(* Logix 5000 project; controller Brake_System vendor 1 type 14 code 242 rev 32.11; software revision 32.00 *)

TASK MainTask (continuous, watchdog 500 ms) : MainProgram
TASK SafetyTask (periodic, rate 20 ms, priority 10, watchdog 20 ms, safety) : SafetyProgram

MODULES
   Local : vendor 1 type 14 code 242 (5069 0, rev 32.11)
END_MODULES

PROGRAM MainProgram   (* main routine MainRoutine *)

ROUTINE MainRoutine   (* ladder *)
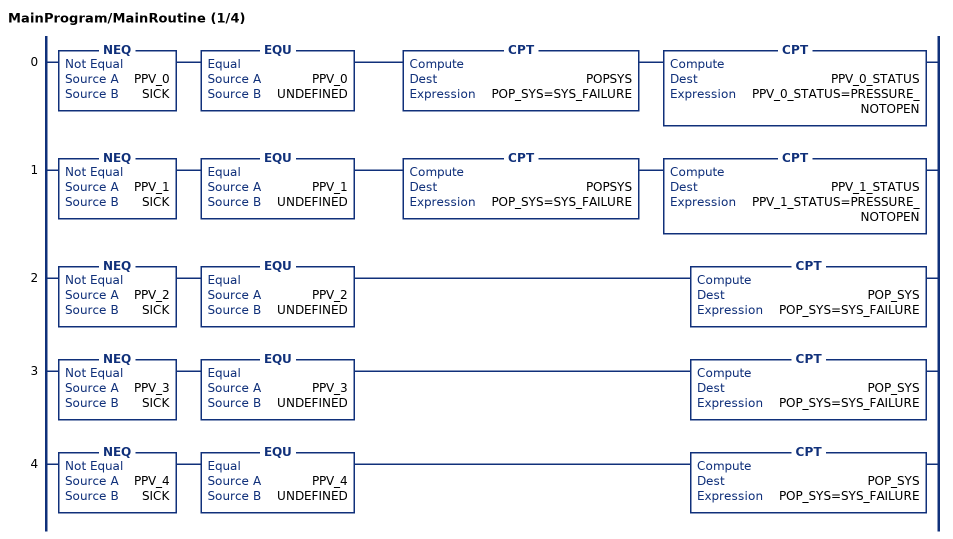
   0: NEQ(PPV_0,SICK)EQU(PPV_0,UNDEFINED)CPT(POPSYS,POP_SYS=SYS_FAILURE)CPT(PPV_0_STATUS,PPV_0_STATUS=PRESSURE_NOTOPEN);
   1: NEQ(PPV_1,SICK)EQU(PPV_1,UNDEFINED)CPT(POPSYS,POP_SYS=SYS_FAILURE)CPT(PPV_1_STATUS,PPV_1_STATUS=PRESSURE_NOTOPEN);
   2: NEQ(PPV_2,SICK)EQU(PPV_2,UNDEFINED)CPT(POP_SYS,POP_SYS=SYS_FAILURE);
   3: NEQ(PPV_3,SICK)EQU(PPV_3,UNDEFINED)CPT(POP_SYS,POP_SYS=SYS_FAILURE);
   4: NEQ(PPV_4,SICK)EQU(PPV_4,UNDEFINED)CPT(POP_SYS,POP_SYS=SYS_FAILURE);
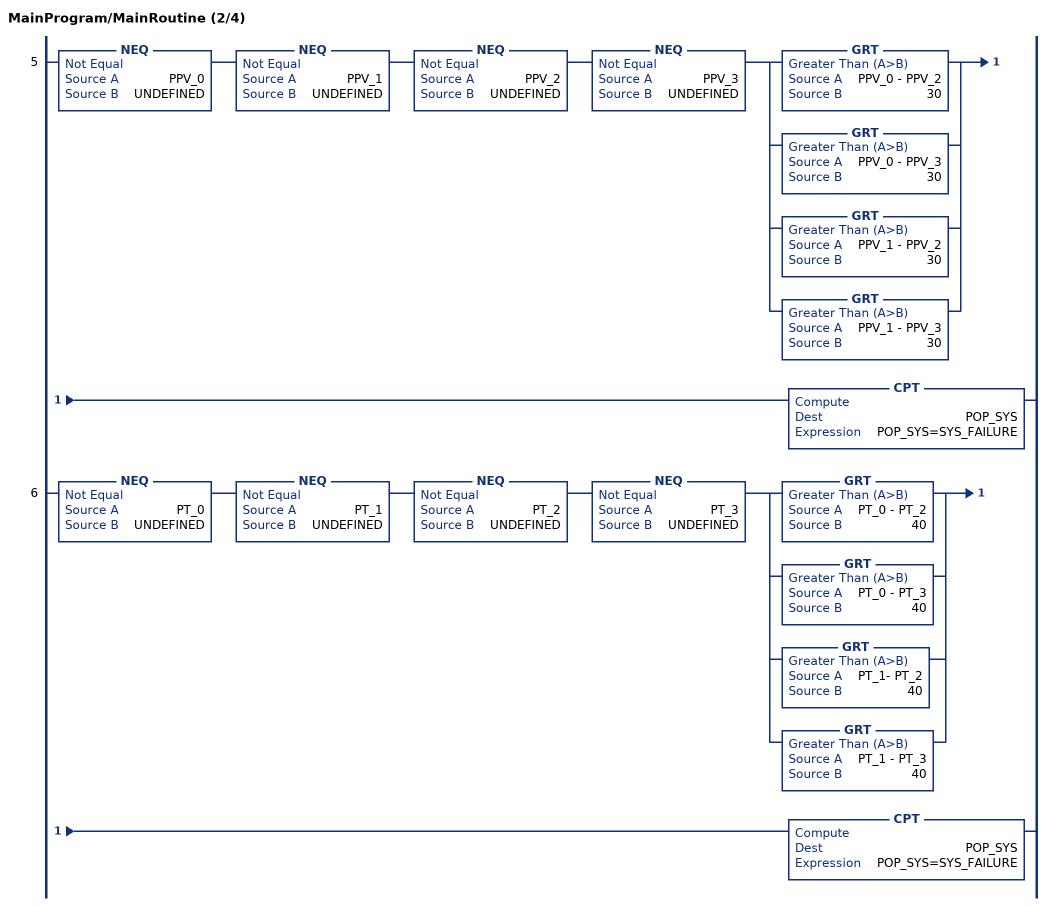
   5: NEQ(PPV_0,UNDEFINED)NEQ(PPV_1,UNDEFINED)NEQ(PPV_2,UNDEFINED)NEQ(PPV_3,UNDEFINED)[GRT(PPV_0 - PPV_2,30) ,GRT(PPV_0 - PPV_3,30) ,GRT(PPV_1 - PPV_2,30) ,GRT(PPV_1 - PPV_3,30) ]CPT(POP_SYS,POP_SYS=SYS_FAILURE);
   6: NEQ(PT_0,UNDEFINED)NEQ(PT_1,UNDEFINED)NEQ(PT_2,UNDEFINED)NEQ(PT_3,UNDEFINED)[GRT(PT_0 - PT_2,40) ,GRT(PT_0 - PT_3,40) ,GRT(PT_1- PT_2,40) ,GRT(PT_1 - PT_3,40) ]CPT(POP_SYS,POP_SYS=SYS_FAILURE);
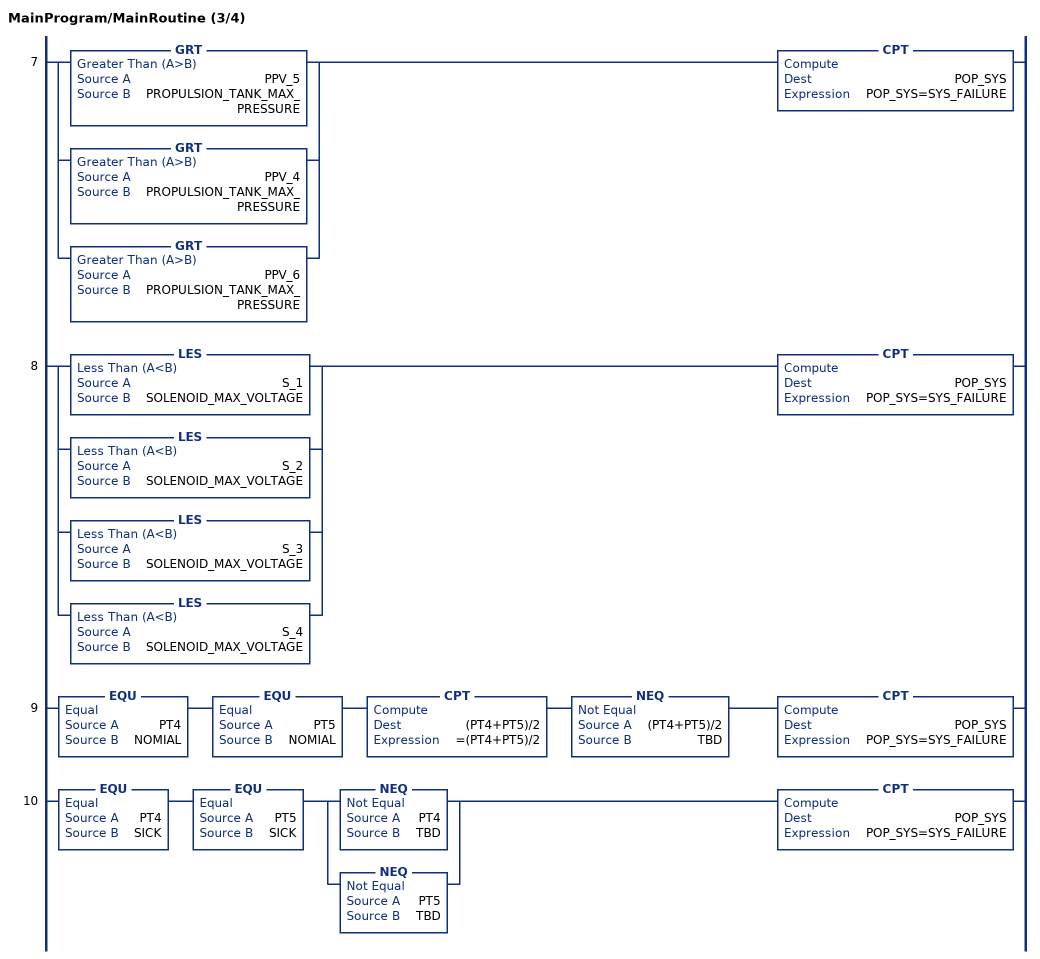
   7: [GRT(PPV_5,PROPULSION_TANK_MAX_PRESSURE) ,GRT(PPV_4,PROPULSION_TANK_MAX_PRESSURE) ,GRT(PPV_6,PROPULSION_TANK_MAX_PRESSURE) ]CPT(POP_SYS,POP_SYS=SYS_FAILURE);
   8: [LES(S_1,SOLENOID_MAX_VOLTAGE) ,LES(S_2,SOLENOID_MAX_VOLTAGE) ,LES(S_3,SOLENOID_MAX_VOLTAGE) ,LES(S_4,SOLENOID_MAX_VOLTAGE) ]CPT(POP_SYS,POP_SYS=SYS_FAILURE);
   9: EQU(PT4,NOMIAL)EQU(PT5,NOMIAL)CPT((PT4+PT5)/2,=(PT4+PT5)/2)NEQ((PT4+PT5)/2,TBD)CPT(POP_SYS,POP_SYS=SYS_FAILURE);
   10: EQU(PT4,SICK)EQU(PT5,SICK)[NEQ(PT4,TBD) ,NEQ(PT5,TBD) ]CPT(POP_SYS,POP_SYS=SYS_FAILURE);
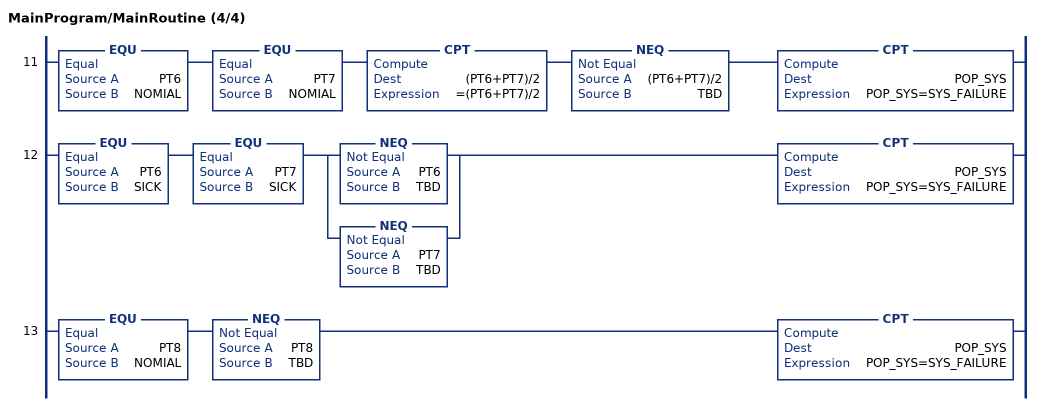
   11: EQU(PT6,NOMIAL)EQU(PT7,NOMIAL)CPT((PT6+PT7)/2,=(PT6+PT7)/2)NEQ((PT6+PT7)/2,TBD)CPT(POP_SYS,POP_SYS=SYS_FAILURE);
   12: EQU(PT6,SICK)EQU(PT7,SICK)[NEQ(PT6,TBD) ,NEQ(PT7,TBD) ]CPT(POP_SYS,POP_SYS=SYS_FAILURE);
   13: EQU(PT8,NOMIAL)NEQ(PT8,TBD)CPT(POP_SYS,POP_SYS=SYS_FAILURE);
END_ROUTINE
END_PROGRAM

PROGRAM SafetyProgram   (* main routine MainRoutine, safety *)

ROUTINE MainRoutine   (* ladder *)
END_ROUTINE
END_PROGRAM
